FUNCTION_BLOCK DT_TO_TD_UINT (* Converts DATE_AND_TIME to TD and DOY *)
  (* Standard: 61499-2; Description: Converts DATE_AND_TIME to TD (time of day in s since 00:00:00.000 [0,..1439]) and DOY (day of the year [1,..,365]) *)
  (* Version 1.0, 2017-06-05, Marc Jakobi, HTW Berlin *)
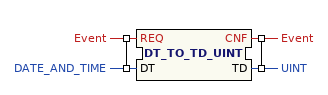
  EVENT_INPUT
    REQ WITH DT; (* Normal Execution Request *)
  END_EVENT
  EVENT_OUTPUT
    CNF WITH TD; (* Execution Confirmation *)
  END_EVENT
  VAR_INPUT
    DT : DATE_AND_TIME; (* Input date *)
  END_VAR
  VAR_OUTPUT
    TD : UINT; (* Time of day in s [0,..,1439] *)
  END_VAR
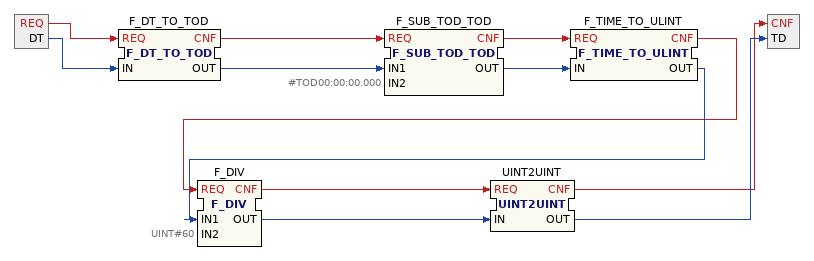
  FBS
    F_DT_TO_TOD : F_DT_TO_TOD;
    F_SUB_TOD_TOD : F_SUB_TOD_TOD(IN2 := #TOD00:00:00.000);
    F_DIV : F_DIV(IN2 := UINT#60);
    UINT2UINT : UINT2UINT;
    F_TIME_TO_ULINT : F_TIME_TO_ULINT;
  END_FBS
  EVENT_CONNECTIONS
    F_DT_TO_TOD.CNF TO F_SUB_TOD_TOD.REQ;
    REQ TO F_DT_TO_TOD.REQ;
    F_DIV.CNF TO UINT2UINT.REQ;
    UINT2UINT.CNF TO CNF;
    F_SUB_TOD_TOD.CNF TO F_TIME_TO_ULINT.REQ;
    F_TIME_TO_ULINT.CNF TO F_DIV.REQ;
  END_CONNECTIONS
  DATA_CONNECTIONS
    F_DT_TO_TOD.OUT TO F_SUB_TOD_TOD.IN1;
    DT TO F_DT_TO_TOD.IN;
    F_DIV.OUT TO UINT2UINT.IN;
    UINT2UINT.OUT TO TD;
    F_SUB_TOD_TOD.OUT TO F_TIME_TO_ULINT.IN;
    F_TIME_TO_ULINT.OUT TO F_DIV.IN1;
  END_CONNECTIONS
END_FUNCTION_BLOCK
